# EPICS StreamDevice protocol: CavitySimulator-loc/CavitySimulatorApp/Db/Temperature.proto
# Protocols for temperature

ExtraInput = Ignore;

InTerminator = NL;
OutTerminator = NL "*OPC?" NL;

getTemp { out "MEAS:TEMP:\$1?"; in "%(\$2:CavitySimulator:Temp\$1Result.VAL)f";}
